// TwinCAT 3 PLC project BufferTest
// ProgramVersion: 3.1.4024.0
// libraries:
//   Tc2_Standard, * (Beckhoff Automation GmbH)
//   Tc2_System, * (Beckhoff Automation GmbH)
//   Tc2_Utilities, * (Beckhoff Automation GmbH)
//   Tc3_Module, * (Beckhoff Automation GmbH)
// project tree:
//   DUTs/ ST_Event.TcDUT, E_EventType.TcDUT
//   / PlcTask.TcTTO
//   POUs/ FB_EventBuffer.TcPOU, MAIN.TcPOU
// real-time tasks:
//   TASK PlcTask: cycle T#10ms, priority 20, ADS port 350
//   TASK PlcTask1: cycle T#10ms, priority 21, ADS port 351

CONFIGURATION BufferTest
    RESOURCE PLC ON TwinCAT3
        TASK PlcTask(INTERVAL := T#10ms, PRIORITY := 20);
        PROGRAM MAIN WITH PlcTask : MAIN;
    END_RESOURCE
END_CONFIGURATION

// ---- DUTs/ST_Event.TcDUT
TYPE ST_Event :
STRUCT
	eEventType : E_EventType;
	eEventSeverity : TcEventSeverity;
	nEventIdentity : UDINT;
	sEventText : STRING(255);
	dtTimestamp : DATE_AND_TIME;
END_STRUCT
END_TYPE

// ---- DUTs/E_EventType.TcDUT
{attribute 'qualified_only'}
{attribute 'strict'}
{attribute 'to_string'}
TYPE E_EventType :
(
	Alarm := 0,
	Message := 1
);
END_TYPE

// ---- POUs/MAIN.TcPOU
PROGRAM MAIN
VAR
	EventBuffer : FB_EventBuffer;
	
	bAddEvent : BOOL;
	stEventToAdd : ST_Event;
	bEventToAddError : BOOL;
	
	
	bReadAndRemoveEvent : BOOL;
	stLastReadEvent : ST_Event;
	bLastEventToReadError : BOOL;
END_VAR

IF bAddEvent THEN
	EventBuffer.AddEvent(stEvent := stEventToAdd, bError => bEventToAddError);
	bAddEvent := FALSE;
END_IF
IF bReadAndRemoveEvent THEN
	EventBuffer.GetAndRemoveEvent(stEvent => stLastReadEvent, bError => bLastEventToReadError);
	bReadAndRemoveEvent := FALSE;
END_IF

END_PROGRAM

// ---- POUs/FB_EventBuffer.TcPOU
FUNCTION_BLOCK FB_EventBuffer
VAR
    MemRingBuffer : FB_MemRingBuffer;
	BufferArray : ARRAY[0..MAX_BUFFER_SIZE] OF BYTE;
END_VAR
VAR CONSTANT
	SIZE_OF_ST_EVENT : UDINT := SIZEOF(ST_Event);
	MAX_NUMBER_OF_ST_EVENTS : UDINT := 5;
	MAX_BUFFER_SIZE : UDINT := SIZE_OF_ST_EVENT * MAX_NUMBER_OF_ST_EVENTS + SIZEOF(MemRingBuffer);
END_VAR

METHOD PUBLIC AddEvent
VAR_INPUT
	stEvent : REFERENCE TO ST_Event;
END_VAR
VAR_OUTPUT
	bError : BOOL;
END_VAR
MemRingBuffer.A_AddTail(pWrite := ADR(stEvent), 
						cbWrite := SIZEOF(stEvent), 
						pBuffer := ADR(BufferArray), 
						cbBuffer := SIZEOF(BufferArray));
						
bError := NOT MemRingBuffer.bOk;
END_METHOD

METHOD PUBLIC GetAndRemoveEvent
VAR_OUTPUT
	stEvent : ST_Event;
	bError : BOOL;
END_VAR
MemRingBuffer.A_RemoveHead(pRead := ADR(stEvent), cbRead := SIZEOF(stEvent), pBuffer := ADR(BufferArray), cbBuffer := SIZEOF(BufferArray));
						
bError := NOT MemRingBuffer.bOk;
END_METHOD

END_FUNCTION_BLOCK
